FUNCTION_BLOCK EventLogger
VAR
	EventBuffer : ARRAY[1..MAXIMUM_SIZE_OF_EVENT_BUFFER] OF ST_Event;
	CurrentEventBufferIndex : INT := 0;
END_VAR
VAR CONSTANT
	MAXIMUM_SIZE_OF_EVENT_BUFFER : INT := 100;
END_VAR

(*Returns TRUE if add was succesful and FALSE if buffer is full*)
METHOD AddEvent : BOOL
VAR_INPUT
	eEventType : E_EventType;
	eEventSeverity : TcEventSeverity;
	nEventIdentity : UDINT;
	sEventText: STRING(255);
END_VAR
IF IsEventBufferFull() THEN
	CurrentEventBufferIndex := CurrentEventBufferIndex + 1;
	EventBuffer[CurrentEventBufferIndex].eEventType := eEventType;
	EventBuffer[CurrentEventBufferIndex].eEventSeverity := eEventSeverity;
	EventBuffer[CurrentEventBufferIndex].nEventIdentity := nEventIdentity;
	EventBuffer[CurrentEventBufferIndex].sEventText := sEventText;
	UpdateEventTimeStampWithSystemTime(stEvent := EventBuffer[CurrentEventBufferIndex]);
	AddEvent:= TRUE;
ELSE
	AddEvent:= FALSE;
END_IF
END_METHOD

METHOD PRIVATE IsEventBufferFull : BOOL
IF (CurrentEventBufferIndex + 1) > MAXIMUM_SIZE_OF_EVENT_BUFFER THEN
	IsEventBufferFull := TRUE;
ELSE
	IsEventBufferFull := FALSE;
END_IF
END_METHOD

END_FUNCTION_BLOCK

(* stored: Version 1.1.0.1, ProductVersion 3.1.4024.5
   POU EventLogger: Id {efc3729f-9194-4f55-accb-e128a3a93159}, SpecialFunc None
   Method AddEvent: Id {aa621d95-f86f-47f7-a615-6760a84f8f28}
   Method IsEventBufferFull: Id {53ddb093-8e5e-47aa-b71a-e74f659a2f30} *)
